Staubli VAL3: Simulation.pjx

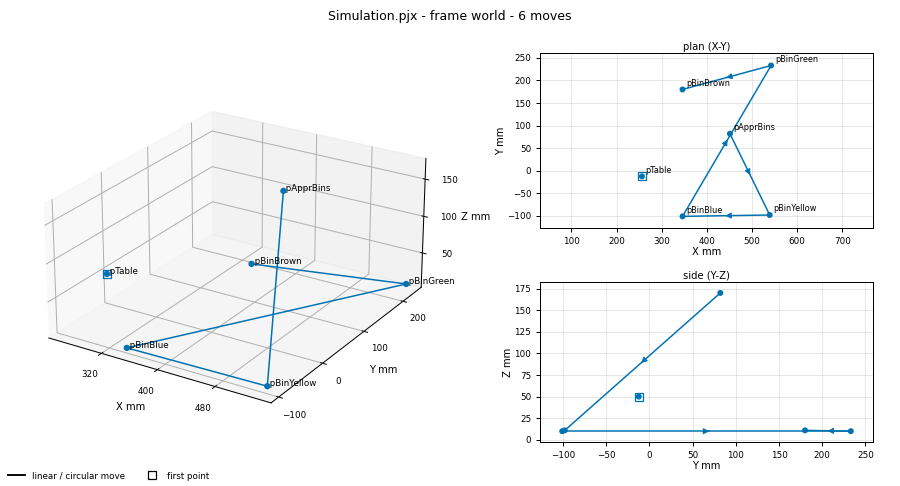
[picture p0: tool path of Simulation.pjx in frame world, 6 of 14 moves have a stored position in this frame; points joined in program order, loops and branches not executed]
--- Simulation.pjx ---
Parameters version=s7.11.2 stackSize=5000 millimeterUnit=true
Program file=moveRobot.pgx
Program file=moveRobotSuc.pgx
Program file=pantalla.pgx
Program file=start.pgx
Program file=startingSockets.pgx
Program file=statesRobot.pgx
Program file=stop.pgx
Data file=Simulation.dtx

--- Simulation.dtx ---
mdesc mNomSpeed
sio sSocket = {link=Socket\Feedback}
tool tToolSuccion = {z=110, fatherId=flange[0], ioLink=valve2}
num nConnection
num nRecvData
jointRx JApproach1 = {j2=9, j3=75, j5=93, j6=142}
jointRx JHome = {j3=0.6}
screen sMonitor
num l_nRetVal
pointRx pApprBins = {x=451, y=82, z=170, rx=-178, rz=-39, fatherId=world[0]}
pointRx pBinYellow = {x=539, y=-98, z=11, rx=-178, rz=-39, fatherId=world[0]}
pointRx pBinBlue = {x=346, y=-101, z=10, rx=-178, rz=-39, fatherId=world[0]}
pointRx pBinGreen = {x=542, y=233, z=10, rx=-178, rz=-39, fatherId=world[0]}
pointRx pBinBrown = {x=346, y=180, z=11, rx=-178, rz=-39, fatherId=world[0]}
jointRx jGetCinta = {j1=-88, j2=71, j3=56, j5=53, j6=50}
bool bStop
num nkey
jointRx jAproachCinta = {j1=-82, j2=60, j3=56.5, j5=65, j6=50}
pointRx pTable = {x=256.13, y=-12.37, z=50, rx=-178, rz=-39, fatherId=world[0]}
tool tToolGripper = {z=115, fatherId=flange[0], ioLink=valve1}
sio sPlc = {link=Socket\PLClient}
num nRecvPLC
jointRx jGetPaperCinta = {j1=-94, j2=83, j3=43, j5=56}
jointRx jGetPlaGlaCinta = {j1=-93, j2=73, j3=54, j5=55}
jointRx jBinGreen = {j1=16, j2=62, j3=30, j5=88, j6=157}
jointRx jBinYellow = {j1=-13, j2=56, j3=41, j5=84, j6=127}
bool bChangeTool
string sTecla
jointRx jChangeTool = {j1=80, j2=45, j3=64, j5=34, j6=52}

--- moveRobotSuc.pgx ---
program moveRobotSuc()
begin
  movej(JHome,tToolSuccion, mNomSpeed)
  waitEndMove()
  movej(JApproach1,tToolSuccion, mNomSpeed)
  waitEndMove()
  do
    movel(pTable,tToolSuccion, mNomSpeed)
    waitEndMove()
    sioGet(sPlc, nRecvPLC)
    if nRecvPLC == 100
      sioSet(sSocket, 82)
      movej(jAproachCinta, tToolSuccion, mNomSpeed)
      waitEndMove()
      movej(jGetCinta, tToolSuccion, mNomSpeed)
      waitEndMove()
      close(tToolSuccion)
      waitEndMove()
      nConnection = sioGet(sSocket, nRecvData)
      switch nRecvData
        case 48
          movej(jGetPlaGlaCinta, tToolSuccion, mNomSpeed)
          waitEndMove()
        break
        case 49
          movej(jGetPaperCinta, tToolSuccion, mNomSpeed)
          waitEndMove()
        break
        case 50
          movej(jGetPlaGlaCinta, tToolSuccion, mNomSpeed)
          waitEndMove()
        break
        case 51
          movej(jGetPlaGlaCinta, tToolSuccion, mNomSpeed)
          waitEndMove()
        break
        default
          putln("Bin selected no correct")
          break
      endSwitch
      movel(pApprBins, tToolSuccion, mNomSpeed)
      waitEndMove()
      switch nRecvData
        case 48
          movel(pBinYellow, tToolSuccion, mNomSpeed)
          waitEndMove()
        break
        case 49
          movel(pBinBlue, tToolSuccion, mNomSpeed)
          waitEndMove()
        break
        case 50
          movel(pBinGreen, tToolSuccion, mNomSpeed)
          waitEndMove()
        break
        case 51
          movel(pBinBrown, tToolSuccion, mNomSpeed)
          waitEndMove()
        break
        default
          putln("Bin selected no correct")
        break
      endSwitch
      open(tToolSuccion)
      waitEndMove()
      nRecvPLC=0
      clearBuffer(sPlc)
    endIf
  until 1==2
end

--- pantalla.pgx ---
program pantalla()
begin
  userPage()
  cls()
  title("Start to recicling")
  gotoxy(35,13)
  put("EXIT")
  do
    gotoxy(0,6)
    //put("Value PLC:")
    //putln(nRecvPLC)
    gotoxy(0,1)
    put("Port 11001:")
    gotoxy(12,1)
    switch nConnection
      case -1
        put("Waiting connection")
      break
      case 1
        putln("Connected succesful")
        put("Go to bin: ")
        switch nRecvData
          case 48
            putln("Yellow")
          break
          case 49
            putln("Blue")
          break
          case 50
            putln("Green")
          break
          case 51
            putln("Brown")
          break
          default
            putln("Bin selected no correct")
          break
        endSwitch
      break
      case 0
        putln("Stopped Connection")
      break
      default
        put("Connection lose")
      break
    endSwitch
  until 1==2
end
